PROGRAM P_Outputs_Laptop
VAR
	//
	n_temp_speed_SP1: REAL;
	n_temp_speed_AP1: REAL;
	n_temp_speed_MI1: REAL;
	
	n_temp_speed_CP1: REAL;
	n_temp_flowrate_CP1: REAL;
	
	
	// temp data for concrete pump
	n_max_pump_speed: REAL :=75; // by measure 
	n_target_pump_speed: REAL :=25; // by calibration (7.5L/min)
	n_test_pump_speed: REAL :=50; // by (15L/min) 0.3 L/rev
END_VAR

//***********************************************************************************
//
// ETH Zürich / Robotic Fabrication Lab
// HIB C 13 / Stefano-Franscini-Platz 1
// CH-8093 Zürich
// 
// ***********************************************************************************
// 
// PROJECT     :  A061 Digital Casting System
// 
// FUNCTION    :  Outputs Laptop Mode
// 
// AUTHOR      :  Weiting Chen/ Philippe Fleischmann 
// 
// EMAIL       :  chenw@usi.ch
// 
// Copyright   :  USI , ETH Zürich (CH) 2022
//
// ***********************************************************************************


//***********************************************************************************
// Mixer 1
//***********************************************************************************

// pass

//***********************************************************************************
// Superplasticizer pump 1
//***********************************************************************************

//
// Power on
GVL_IO.ob_SP1_Power_On:=GVL_VAR.b_Mode_Laptop;
//
// Pressure is Okay, always set it to True
GVL_IO.ob_SP1_Pressure_Ok:=TRUE;
//
// Bucket is not empty, always set it to true
GVL_IO.ob_SP1_Not_Empty:=TRUE;
//
// Pulse mode is a preset amount,  not in use
GVL_IO.ob_SP1_Pulse:=FALSE;


//
// Start pump
IF		P_SP1_OnOff.n_step= 30 
	OR 	P_SP1_Check.n_Step= 30 
THEN
	//
	// Pump On
	GVL_IO.ob_SP1_Start:=TRUE;
ELSE
	//
	// Pump On
	GVL_IO.ob_SP1_Start:=FALSE;
END_IF

//
// Speeds for Superplastizier pump
IF GVL_ResearchData.b_RED_Superplasticizer_Pump_Flush_On AND P_SP1_OnOff.n_step= 30 THEN
	//
	// Process speed for flushing or filling the pipe
	n_temp_speed_SP1:=GVL_ResearchData.n_RED_Superplasticizer_Pump_Flush_Flowrate;

ELSIF P_SP1_Check.n_Step=20 OR P_SP1_Check.n_Step=30 THEN 	
	//	
	// Check Flowrate for pump
	n_temp_speed_SP1:=GVL_ResearchData.n_RED_Superplasticizer_Pump_Check_Flowrate;
	
ELSE
	//
	// Process speed for pump
	n_temp_speed_SP1:=GVL_ResearchData.n_RED_Superplasticizer_Pump_Flowrate;

END_IF

GVL_IO.on_SP1_Speed:=F_ScalAnalogOut(
	n_Input:= REAL_TO_INT(n_temp_speed_SP1),
	n_InMin:= 0, 
	n_InMax:= REAL_TO_INT(GVL_ResearchData.f_RED_Status_Superplasticizer_Pump_Max_Flowrate_ml_per_min), 
	n_OutMin:= 0, 
	n_OutMax:= 32767);


//***********************************************************************************
// Accelerator pump 1
//***********************************************************************************

//
// Power on
GVL_IO.ob_AP1_Power_On:=GVL_VAR.b_Mode_Laptop;
//
// Pressure okey always set to true
GVL_IO.ob_AP1_Pressure_Ok:=TRUE;
//
// Bucket not empty always set to true
GVL_IO.ob_AP1_Not_Empty:=TRUE;
//
// Pulse a preset amount not in use
GVL_IO.ob_AP1_Pulse:=FALSE;

//
// Start pump
IF 	   P_AP1_OnOff.n_Step=30 
	OR P_AP1_Check.n_Step=30
THEN
	//
	// Pump on
	GVL_IO.ob_AP1_Start:=TRUE;
ELSE
	//
	// Pump off
	GVL_IO.ob_AP1_Start:=FALSE;
END_IF

//
// Speed for accelerator pump
IF GVL_ResearchData.b_RED_Acceleration_Pump_Flush_On AND P_AP1_OnOff.n_Step=30 THEN
	//
	// Process speed for flushing or filling the pipe
	n_temp_speed_AP1:=GVL_ResearchData.n_RED_Acceleration_Pump_Flush_Flowrate;
ELSIF P_AP1_Check.n_Step=20 OR P_AP1_Check.n_Step=30 THEN
	//	
	// Check Flowrate for pump
	n_temp_speed_AP1:=GVL_ResearchData.n_RED_Acceleration_Pump_Check_Flowrate;
ELSE
	//
	// Process speed for pump
	n_temp_speed_AP1:=GVL_ResearchData.n_RED_Acceleration_Pump_Flowrate;
END_IF

GVL_IO.on_AP1_Speed:=F_ScalAnalogOut(
	n_Input:= REAL_TO_INT(n_temp_speed_AP1),
	n_InMin:= 0, 
	n_InMax:= REAL_TO_INT(GVL_ResearchData.f_RED_Status_Acceleration_Pump_Max_Flowrate_ml_per_min), 
	n_OutMin:= 0, 
	n_OutMax:= 32767);


// ***********************************************************************************
// Concrete Pump 1 
// ***********************************************************************************

//
// Start
IF  P_CP1_Enable.n_Step=20 THEN
	GVL_IO.ob_CP1_Start:=TRUE;
ELSE
	GVL_IO.ob_CP1_Start:=FALSE;
END_IF

//
// Stop
IF  P_CP1_Enable.n_Step=40 THEN
	GVL_IO.ob_CP1_Stop:=TRUE;
ELSE
	GVL_IO.ob_CP1_Stop:=FALSE;
END_IF


//
// Forward
GVL_IO.ob_CP1_Forward:=GVL_ResearchData.b_RED_Concrete_Pump_Forward_On;

//
// Backward
GVL_IO.ob_CP1_Backward:=GVL_ResearchData.b_RED_Concrete_Pump_Backward_On;

//
// Concrete pump speed  0 (0V) to 75 rpm (10V)
// Concrete pump max target speed  0 to 25 rpm
// Concrete pump max target Flowrate  0 to 5000 ml/min
// Theoretic Dosing Volume for Concrete pump is 200 ml/rev 

IF GVL_ResearchData.b_RED_Concrete_Pump_Flush_On THEN
	//
	// Process speed for flushing or filling the pipe
	n_temp_flowrate_CP1:=GVL_ResearchData.f_RED_Status_Concrete_Pump_Max_Flowrate_l_per_min*1000;
ELSIF P_CP1_Check.n_Step=20 OR P_CP1_Check.n_Step=25 THEN
	//	
	// Check Flowrate for pump
	n_temp_flowrate_CP1:=GVL_ResearchData.f_RED_Concrete_Pump_Check_Flowrate*1000;
ELSE
	//
	// Process speed for pump
	n_temp_flowrate_CP1:=GVL_ResearchData.f_RED_Concrete_Pump_Flowrate*1000;
END_IF


// temporary remapping  
n_temp_speed_CP1:=F_Mapping_REAL(
	f_Input:= n_temp_flowrate_CP1, 
	f_InMin:= 0, 
	f_InMax:= 15*1000, 
	f_OutMin:= 0, 
	f_OutMax:= n_test_pump_speed);

// Concrete pump speed  0 (0V) to 75 rpm (10V)
GVL_IO.on_CP1_Speed:=REAL_TO_INT(F_Mapping_REAL(
	f_Input:= n_temp_speed_CP1, 
	f_InMin:= 0, 
	f_InMax:= n_max_pump_speed, 
	f_OutMin:= 0, 
	f_OutMax:= 32767));

END_PROGRAM

(* stored: Version 1.1.0.1, ProductVersion 3.1.4024.2
   POU P_Outputs_Laptop: Id {bcd714bb-3f40-4b88-8117-548c3a821447}, SpecialFunc None *)
